(* CODESYS project MT6_Decoiler2.project

Project tree, tasks and I/O mapping:
  PLC_AC500 : AC500 PM564-ETH, ABB Automation Products GmbH, order no. 1SAP12xx00R0071, version 2.8.0.0
      settings: PM5xx Type = PM564-ETH; CoDeSys V2.3 Target = 23846; Checksum = 0; Checksum-PLC = 0; Product version = [2, 2, 0, 4]
    Application
      application App
    OBIO : 6DI+6DO+2AI+1AO, ABB Automation Products GmbH, version 2.8.0.0
        input  iStop : BOOL  // Digital inputs DI0 - DI5, AI0 - AI1.Digital input DI0
        input  iStart : BOOL  // Digital inputs DI0 - DI5, AI0 - AI1.Digital input DI1
        input  iUnwindFwd : BOOL  // Digital inputs DI0 - DI5, AI0 - AI1.Digital input DI2
        input  iUnwindRev : BOOL  // Digital inputs DI0 - DI5, AI0 - AI1.Digital input DI3
        input  iMandrelExpand : BOOL  // Digital inputs DI0 - DI5, AI0 - AI1.Digital input DI4
        input  iMandrelCollapse : BOOL  // Digital inputs DI0 - DI5, AI0 - AI1.Digital input DI5
        input  iwLoopSensor : INT  // Analog input AI0
        output qUnwinderFwd : BOOL  // Digital outputs DO0 / NO0 - DO5 / NO5.Digital output DO0 / NO0
        output qUnwinderRev : BOOL  // Digital outputs DO0 / NO0 - DO5 / NO5.Digital output DO1 / NO1
        output qPinchRollUp : BOOL  // Digital outputs DO0 / NO0 - DO5 / NO5.Digital output DO2 / NO2
        output qPinchRollDown : BOOL  // Digital outputs DO0 / NO0 - DO5 / NO5.Digital output DO3 / NO3
        output qThreadingUp : BOOL  // Digital outputs DO0 / NO0 - DO5 / NO5.Digital output DO4 / NO4
        output qThreadingDown : BOOL  // Digital outputs DO0 / NO0 - DO5 / NO5.Digital output DO5 / NO5
        output qwDriveRef : INT  // Analog output AOI / AOU
        unmapped channels: Digital inputs DI0 - DI5, AI0 - AI1, Interrupt DI0 - DI3, Analog input AI1, State Byte PWM 2, State Byte PWM 3, Unused, Unused, Unused, Unused, Unused, Unused, Unused, Unused, Unused, Unused, Unused, Unused, Unused, Unused, Actual value 1, Actual value 2, State Byte 1, State Byte 2, Digital outputs DO0 / NO0 - DO5 / NO5, Control Byte PWM 2, PWM 2, frequency / cycle time, PWM 2, duty cycle / duty time, Control Byte PWM 3, Unused, PWM 3, frequency / cycle time, PWM 3, duty cycle / duty time, Unused, Unused, Unused, Unused, Unused, Unused, Unused, Unused, Unused,
          Unused, Unused, Start value 1, End value 1, Start value 2, End value 2, Control Byte 1, Control Byte 2
    IO_Bus : I/O-Bus, ABB Automation Products GmbH, version 2.8.0.0
      DX561_1 : DX561, ABB Automation Products GmbH, order no. 1TNE968902R2301, version 2.8.0.0
          input  iSnubberRollUp : BOOL  // Digital inputs I0 - I7.Digital input I0
          input  iSnubberRollDown : BOOL  // Digital inputs I0 - I7.Digital input I1
          input  iCoilDown : BOOL  // Digital inputs I0 - I7.Digital input I2
          input  iCoilUp : BOOL  // Digital inputs I0 - I7.Digital input I3
          input  iTraverseIn : BOOL  // Digital inputs I0 - I7.Digital input I4
          input  iTraverseOut : BOOL  // Digital inputs I0 - I7.Digital input I5
          input  iBrakeOn : BOOL  // Digital inputs I0 - I7.Digital input I6
          input  iDriveReady : BOOL  // Digital inputs I0 - I7.Digital input I7
          output qMandrelExpand : BOOL  // Digital outputs O0 - O7.Digital output O0
          output qMandrelCollapse : BOOL  // Digital outputs O0 - O7.Digital output O1
          output qSnubberRollUp : BOOL  // Digital outputs O0 - O7.Digital output O2
          output qSnubberRollDown : BOOL  // Digital outputs O0 - O7.Digital output O3
          output qCoilDown : BOOL  // Digital outputs O0 - O7.Digital output O4
          output qCoilUp : BOOL  // Digital outputs O0 - O7.Digital output O5
          output qTraverseIn : BOOL  // Digital outputs O0 - O7.Digital output O6
          output qTraverseOut : BOOL  // Digital outputs O0 - O7.Digital output O7
          unmapped channels: Digital inputs I0 - I7, Digital outputs O0 - O7, Digital inputs I0 - I7, Digital outputs O0 - O7, Digital inputs I0 - I7, Digital outputs O0 - O7
      DX561 : DX561, ABB Automation Products GmbH, order no. 1TNE968902R2301, version 2.8.0.0
          input  iPinchRollUp : BOOL  // Digital inputs I0 - I7.Digital input I0
          input  iPinchRollDown : BOOL  // Digital inputs I0 - I7.Digital input I1
          input  iThreadingUp : BOOL  // Digital inputs I0 - I7.Digital input I2
          input  iThreadingDown : BOOL  // Digital inputs I0 - I7.Digital input I3
          input  iAuto : BOOL  // Digital inputs I0 - I7.Digital input I4
          input  iUnwinderTrip : BOOL  // Digital inputs I0 - I7.Digital input I5
          input  iStraightnerInchFwd : BOOL  // Digital inputs I0 - I7.Digital input I6
          input  iStraightnerInchRev : BOOL  // Digital inputs I0 - I7.Digital input I7
          output qStartSensing : BOOL  // Digital outputs O0 - O7.Digital output O0
          output qBrakeOn : BOOL  // Digital outputs O0 - O7.Digital output O1
          output qRelieveValve : BOOL  // Digital outputs O0 - O7.Digital output O2
          output qRunIndicator : BOOL  // Digital outputs O0 - O7.Digital output O3
          output qVFDStartFwd : BOOL  // Digital outputs O0 - O7.Digital output O4
          output qVFDStartRev : BOOL  // Digital outputs O0 - O7.Digital output O5
          unmapped channels: Digital inputs I0 - I7, Digital outputs O0 - O7, Digital inputs I0 - I7, Digital outputs O0 - O7, Digital inputs I0 - I7, Digital outputs O0 - O7
    Interfaces : Interfaces, ABB Automation Products GmbH, version 2.8.0.0
      COM1_Modbus : COM1 - Modbus, ABB Automation Products GmbH, version 2.8.0.0
      COM2_None : COM2 - None, ABB Automation Products GmbH, version 2.8.0.0
      Ethernet : Onboard Ethernet, ABB Automation Products GmbH, version 2.8.0.0
        ETH1 : ETH1, ABB Automation Products GmbH, version 2.8.0.0
            settings: Gateway = 3232235521
        Protocols : Protocols, ABB Automation Products GmbH, version 2.8.0.0
  program POU [FBD]
  global variables GVL
  program Outputs [FBD]
*)

// GVL
VAR_GLOBAL
END_VAR

// POU
PROGRAM POU
VAR
END_VAR

// NETWORK 1

END_PROGRAM

// Outputs
PROGRAM Outputs
VAR
END_VAR

// NETWORK 1

END_PROGRAM
